// Mitsubishi GX Works2 project: 2   PLC: Q02/Q02H
// 2

PROGRAM MAIN
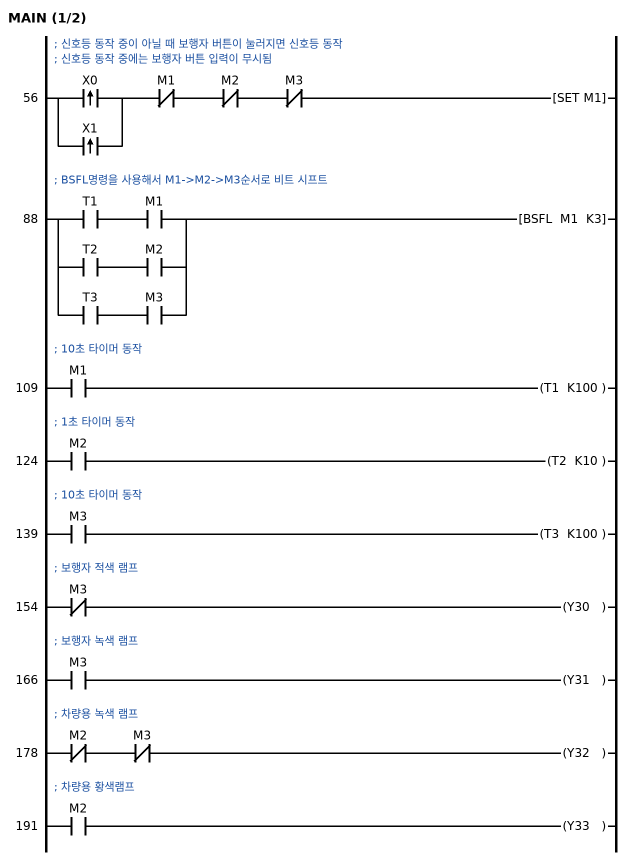
; 신호등 동작 중이 아닐 때 보행자 버튼이 눌러지면 신호등 동작
; 신호등 동작 중에는 보행자 버튼 입력이 무시됨
56    LDP     X0
      ORP     X1
      ANI     M1
      ANI     M2
      ANI     M3
      SET     M1
; BSFL명령을 사용해서 M1->M2->M3순서로 비트 시프트
88    LD      T1
      AND     M1
      LD      T2
      AND     M2
      ORB
      LD      T3
      AND     M3
      ORB
      BSFL    M1 K3
; 10초 타이머 동작
109   LD      M1
      OUT     T1 K100
; 1초 타이머 동작
124   LD      M2
      OUT     T2 K10
; 10초 타이머 동작
139   LD      M3
      OUT     T3 K100
; 보행자 적색 램프
154   LDI     M3
      OUT     Y30
; 보행자 녹색 램프
166   LD      M3
      OUT     Y31
; 차량용 녹색 램프
178   LDI     M2
      ANI     M3
      OUT     Y32
; 차량용 황색램프
191   LD      M2
      OUT     Y33
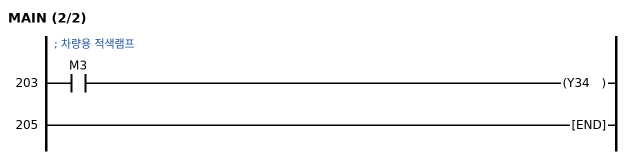
; 차량용 적색램프
203   LD      M3
      OUT     Y34
205   END
END_PROGRAM
